Fanuc TP program (LS listing): bg_hmi_messages.ls

/PROG  BG_HMI_MESSAGES
/ATTR
OWNER		= MNEDITOR;
COMMENT		= "";
PROG_SIZE	= 4483;
CREATE		= DATE 23-11-18  TIME 09:11:50;
MODIFIED	= DATE 24-03-05  TIME 13:03:38;
FILE_NAME	= ;
VERSION		= 0;
LINE_COUNT	= 167;
MEMORY_SIZE	= 4859;
PROTECT		= READ_WRITE;
TCD:  STACK_SIZE	= 0,
      TASK_PRIORITY	= 50,
      TIME_SLICE	= 0,
      BUSY_LAMP_OFF	= 0,
      ABORT_REQUEST	= 0,
      PAUSE_REQUEST	= 0;
DEFAULT_GROUP	= 1,*,*,*,*;
CONTROL_CODE	= 00000000 00000000;
/APPL
/APPL

AUTO_SINGULARITY_HEADER;
  ENABLE_SINGULARITY_AVOIDANCE   : TRUE;
/MN
   1:  !******************************** ;
   2:  !CONTROLS MESSAGES ON HMI         ;
   3:  !******************************** ;
   4:  !DISABLE MESSAGES IF START IS PR  ;
   5:  IF (DO[100:START PRESSED]=ON) THEN ;
   6:  F[45:MESSAGE 1]=(OFF) ;
   7:  F[46:MESSAGE 2]=(OFF) ;
   8:  F[47:MESSAGE 3]=(OFF) ;
   9:  F[48:MESSAGE 4]=(OFF) ;
  10:  F[49:MESSAGE 5]=(OFF) ;
  11:  F[50:MESSAGE 6]=(OFF) ;
  12:  F[51:MESSAGE 7]=(OFF) ;
  13:  F[52:MESSAGE 8]=(OFF) ;
  14:  F[53:MESSAGE 9]=(OFF) ;
  15:  F[54:MESSAGE 10]=(OFF) ;
  16:  F[55:MESSAGE 11]=(OFF) ;
  17:  F[56:MESSAGE 12]=(OFF) ;
  18:  F[57:MESSAGE 13]=(OFF) ;
  19:  F[58:MESSAGE 14]=(OFF) ;
  20:  F[59:MESSAGE 15]=(OFF) ;
  21:  F[60:MESSAGE 16]=(OFF) ;
  22:  F[61:MESSAGE 17]=(OFF) ;
  23:  F[62:MESSAGE 18]=(OFF) ;
  24:  F[63:MESSAGE 19]=(OFF) ;
  25:  F[64:MESSAGE 20]=(OFF) ;
  26:  F[65:MESSAGE 21]=(OFF) ;
  27:  F[66:MESSAGE 22]=(OFF) ;
  28:  F[67:MESSAGE 23]=(OFF) ;
  29:  F[68:MESSAGE 24]=(OFF) ;
  30:  F[69:MESSAGE 25]=(OFF) ;
  31:  F[70:MESSAGE 26]=(OFF) ;
  32:  F[71:MESSAGE 27]=(OFF) ;
  33:  F[72:MESSAGE 28]=(OFF) ;
  34:  F[73:MESSAGE 29]=(OFF) ;
  35:  F[74:MESSAGE 30]=(OFF) ;
  36:  F[75:MESSAGE 31]=(OFF) ;
  37:  F[76:MESSAGE 32]=(OFF) ;
  38:  F[77:MESSAGE 33]=(OFF) ;
  39:  F[78:MESSAGE 34]=(OFF) ;
  40:  F[79:MESSAGE 35]=(OFF) ;
  41:  ENDIF ;
  42:  !TABLE CANT BE UNLOCKED WHILE     ;
  43:  !ROBOT IS RUNNING                 ;
  44:  IF (DI[38:TABLE UNLOCK (HMI)]=ON AND UO[10:Busy]=ON AND UO[3:Prg running]=ON AND UO[4:Prg paused]=OFF AND F[45:MESSAGE 1]=OFF AND DO[100:START PRESSED]=OFF),F[45:MESSAGE 1]=(ON) ;
  45:   ;
  46:  !TABLE CANT BE UNLOCKED WHILE     ;
  47:  !ROBOT NOT AT HOME                ;
  48:  IF (DI[38:TABLE UNLOCK (HMI)]=ON AND DO[145:AT HOME]=OFF AND F[46:MESSAGE 2]=OFF AND DO[100:START PRESSED]=OFF),F[46:MESSAGE 2]=(ON) ;
  49:   ;
  50:  !TABLE CANT BE LOCKED WHILE       ;
  51:  !ROBOT NOT AT HOME                ;
  52:  IF (DI[39:TABLE LOCK (HMI)]=ON AND DO[145:AT HOME]=OFF AND F[47:MESSAGE 3]=OFF AND DO[100:START PRESSED]=OFF),F[47:MESSAGE 3]=(ON) ;
  53:   ;
  54:  !TABLE CANT BE UNLOCKED WHILE     ;
  55:  !WHILE NOT IN PLACE               ;
  56:  IF (DI[39:TABLE LOCK (HMI)]=ON AND DO[35:TABLE IN POSITION]=OFF AND F[48:MESSAGE 4]=OFF AND DO[100:START PRESSED]=OFF),F[48:MESSAGE 4]=(ON) ;
  57:   ;
  58:  !CYCLE STOP IS ACTIVE             ;
  59:  IF (DI[31:CYCLE STOP REQ]=ON AND F[49:MESSAGE 5]=OFF AND DO[100:START PRESSED]=OFF),F[49:MESSAGE 5]=(ON) ;
  60:   ;
  61:  !ROBOT IS IN STEPMODE             ;
  62:  IF (DO[30:IN STEP MODE]=ON AND DO[100:START PRESSED]=OFF),F[50:MESSAGE 6]=(ON) ;
  63:   ;
  64:  !MANUAL GRIPPER CONTROLS DISABLE  ;
  65:  IF ((UO[10:Busy]=ON) AND (DI[120:T1 OPEN HMI PB]=ON OR DI[121:T1 CLOSE HMI PB]=ON OR DI[122:T2 OPEN HMI PB]=ON OR DI[123:T2 CLOSE HMI PB]=ON)),F[51:MESSAGE 7]=(ON) ;
  66:   ;
  67:  !PART SETUP BUTTON PRESSED        ;
  68:  IF (DO[112:ROBOT OK TO CHANGEOVER]=OFF AND DO[113:SETUP BUTTON PRESSED]=ON AND DO[100:START PRESSED]=OFF),F[52:MESSAGE 8]=(ON) ;
  69:   ;
  70:  !AIR PRESSURE IS LOW              ;
  71:  IF (DI[8:SYSTEM AIR OK]=OFF AND F[53:MESSAGE 9]=OFF AND DO[100:START PRESSED]=OFF),F[53:MESSAGE 9]=(ON) ;
  72:   ;
  73:  !MACHINE CONTROLLER UNSAFE        ;
  74:  IF (DI[7:MACH CNTRL SAFE]=OFF AND DO[100:START PRESSED]=OFF),F[54:MESSAGE 10]=(ON) ;
  75:   ;
  76:   ;
  77:  !NEW PART ACTIVE FOR A SIDE       ;
  78:  IF (DI[103:NEW PART HMI PB]=ON AND DI[2:TABLE AT B POSITION]=ON),F[55:MESSAGE 11]=(ON) ;
  79:   ;
  80:   ;
  81:  !NEW PART ACTIVE FOR B SIDE       ;
  82:  IF (DI[103:NEW PART HMI PB]=ON AND DI[1:TABLE AT A POSITION]=ON),F[56:MESSAGE 12]=(ON) ;
  83:   ;
  84:  !NEW PART RESET                   ;
  85:  IF (DI[103:NEW PART HMI PB]=ON AND DO[102:NEW PART A]=OFF AND DO[103:NEW PART B]=OFF AND DO[104:NEW PART ACTIVE]=OFF),F[57:MESSAGE 13]=(ON) ;
  86:   ;
  87:  !A SIDE PALLET SETUP COMPLETE     ;
  88:  IF (DI[2:TABLE AT B POSITION]=ON AND DI[47:LOAD COMPLETE HMI]=ON),F[58:MESSAGE 14]=(ON) ;
  89:   ;
  90:  !B SIDE PALLET SETUP COMPLETE     ;
  91:  IF (DI[1:TABLE AT A POSITION]=ON AND DI[47:LOAD COMPLETE HMI]=ON),F[59:MESSAGE 15]=(ON) ;
  92:   ;
  93:  !PALLET SETUP COMPLETE            ;
  94:  IF (DI[45:ABORT LOAD SIDE]=ON),F[60:MESSAGE 16]=(ON) ;
  95:   ;
  96:  !TABLE UNLOCKED                   ;
  97:  IF (DI[38:TABLE UNLOCK (HMI)]=ON),F[61:MESSAGE 17]=(ON) ;
  98:   ;
  99:  !TABLE LOCKED                     ;
 100:  IF (DI[39:TABLE LOCK (HMI)]=ON),F[62:MESSAGE 18]=(ON) ;
 101:   ;
 102:  !OPERATOR ESTOP PRESSED           ;
 103:  IF (DO[95:OPERATOR ESTOP]=ON),F[65:MESSAGE 21]=(ON) ;
 104:   ;
 105:  !TEACH PENDANT ESTOP PRESSED      ;
 106:  IF (DO[96:TP ESTOP]=ON),F[66:MESSAGE 22]=(ON) ;
 107:   ;
 108:  !EXT ESTOP PRESSED                ;
 109:  IF (DO[97:EXTERNAL ESTOP]=ON),F[67:MESSAGE 23]=(ON) ;
 110:   ;
 111:  !ROBOT CRASH                      ;
 112:  IF (R[40:RECOVER START PR]>=65 AND R[40:RECOVER START PR]<=69 AND DO[177:COLLISION]=ON),F[68:MESSAGE 24]=(ON) ;
 113:   ;
 114:  !HEARTBEAT FAULT                  ;
 115:  IF (DO[418:HEARTBEAT FAULT]=ON),F[69:MESSAGE 25]=(ON) ;
 116:   ;
 117:  !MACHINE NOT HOME             ;
 118:  IF (UO[3:Prg running]=ON AND DO[196:DOOR OPEN 1 COM]=ON AND DO[199:MACHINE HOME COM]=OFF AND DO[203:SYSTEM LINK COM]=ON AND DO[204:MACHINE IN AUTO COM]=ON AND DO[205:CYCLE COMPLETE COM]=ON AND
    :  DO[224:ROBOT WAITING]=ON) THEN ;
 119:  F[70:MESSAGE 26]=(ON) ;
 120:  ENDIF ;
 121:   ;
 122:  !MACHINE NEEDS PROGRAM END ;
 123:  IF (UO[3:Prg running]=ON AND DO[196:DOOR OPEN 1 COM]=ON AND DO[199:MACHINE HOME COM]=ON AND DO[203:SYSTEM LINK COM]=ON AND DO[204:MACHINE IN AUTO COM]=ON AND DO[205:CYCLE COMPLETE COM]=OFF AND
    :  DO[224:ROBOT WAITING]=ON) THEN ;
 124:  F[71:MESSAGE 27]=(ON) ;
 125:  ENDIF ;
 126:   ;
 127:  !MACHINE NOT IN AUTO ;
 128:  IF (UO[3:Prg running]=ON AND DO[196:DOOR OPEN 1 COM]=ON AND DO[199:MACHINE HOME COM]=ON AND DO[203:SYSTEM LINK COM]=ON AND DO[204:MACHINE IN AUTO COM]=OFF AND DO[205:CYCLE COMPLETE COM]=ON AND
    :  DO[224:ROBOT WAITING]=ON) THEN ;
 129:  F[72:MESSAGE 28]=(ON) ;
 130:  ENDIF ;
 131:   ;
 132:  !MACHINE NOT IN SYSTEM LINK ;
 133:  IF (UO[3:Prg running]=ON AND DO[196:DOOR OPEN 1 COM]=ON AND DO[199:MACHINE HOME COM]=ON AND DO[203:SYSTEM LINK COM]=OFF AND DO[204:MACHINE IN AUTO COM]=ON AND DO[205:CYCLE COMPLETE COM]=ON AND
    :  DO[224:ROBOT WAITING]=ON) THEN ;
 134:  F[73:MESSAGE 29]=(ON) ;
 135:  ENDIF ;
 136:   ;
 137:  !MACHINE DOOR NOT OPEN ;
 138:  IF (UO[3:Prg running]=ON AND DO[196:DOOR OPEN 1 COM]=OFF AND DO[199:MACHINE HOME COM]=ON AND DO[203:SYSTEM LINK COM]=ON AND DO[204:MACHINE IN AUTO COM]=ON AND DO[205:CYCLE COMPLETE COM]=ON AND
    :  DO[224:ROBOT WAITING]=ON) THEN ;
 139:  F[74:MESSAGE 30]=(ON) ;
 140:  ENDIF ;
 141:   ;
 142:  !ROBOT WAITING FOR MACHINE READY ;
 143:  IF (UO[3:Prg running]=ON AND DO[196:DOOR OPEN 1 COM]=OFF AND DO[199:MACHINE HOME COM]=OFF AND DO[203:SYSTEM LINK COM]=ON AND DO[204:MACHINE IN AUTO COM]=ON AND DO[205:CYCLE COMPLETE COM]=OFF AND
    :  DO[224:ROBOT WAITING]=ON) THEN ;
 144:  F[75:MESSAGE 31]=(ON) ;
 145:  ENDIF ;
 146:   ;
 147:  !MACHINE NOT AUTO OR SYSTEM LINK ;
 148:  IF (UO[3:Prg running]=ON AND DO[196:DOOR OPEN 1 COM]=OFF AND DO[199:MACHINE HOME COM]=ON AND (DO[203:SYSTEM LINK COM]=OFF OR DO[204:MACHINE IN AUTO COM]=OFF) AND DO[205:CYCLE COMPLETE COM]=ON AND
    :  DO[224:ROBOT WAITING]=ON) THEN ;
 149:  F[76:MESSAGE 32]=(ON) ;
 150:  ENDIF ;
 151:   ;
 152:  !TURN OFF MESSAGES IF FAULT       ;
 153:  !RESET IS PRESSED                 ;
 154:  IF (DI[43:ROBOT FAULT RESET]=ON) THEN ;
 155:   ;
 156:  DO[29:UALM MESSAGE ACTIVE]=OFF ;
 157:  F[63:MESSAGE 19]=(ON) ;
 158:  F[64:MESSAGE 20]=(ON) ;
 159:  IF ($SCR.$CHAIN_STAT<>0) THEN ;
 160:  $MCR.$CHAIN_RESET=1 ;
 161:  ENDIF ;
 162:  ENDIF ;
 163:   ;
 164:  IF (DI[43:ROBOT FAULT RESET]=OFF AND DI[33:CYCLE START (HMI)]=OFF) THEN ;
 165:  F[63:MESSAGE 19]=(OFF) ;
 166:  F[64:MESSAGE 20]=(OFF) ;
 167:  ENDIF ;
/POS
/END
